RoboDK station: Estación_kuka_ibero_router.rdk

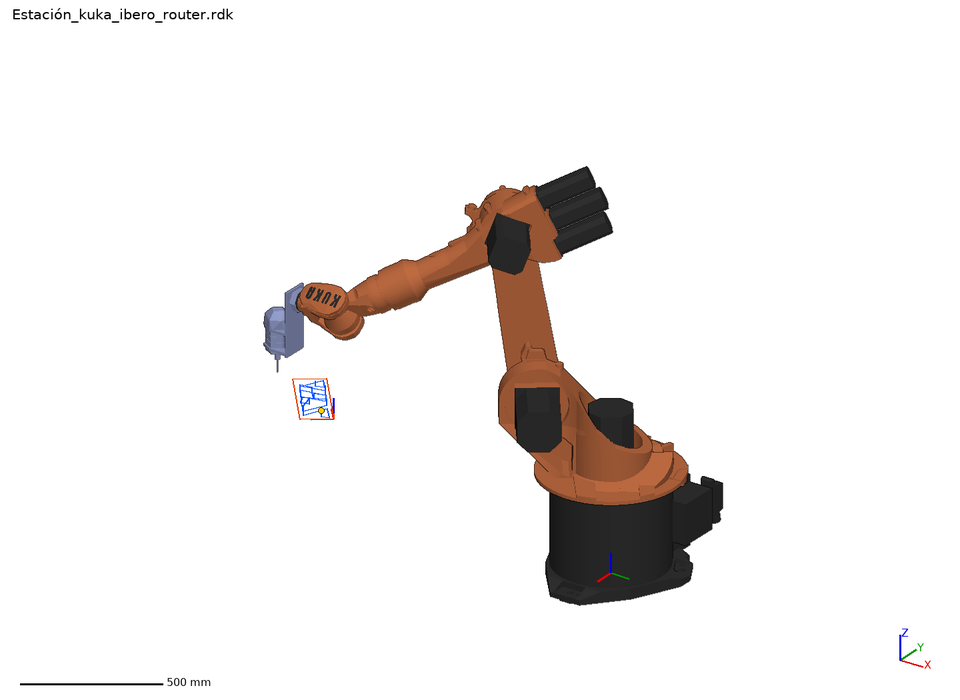
[picture v0: the station drawn from its stored meshes, robots at their saved joint values, targets as dots, program paths as lines]
Station Estación_kuka_ibero_router (saved by RoboDK 5.9.0). Poses are relative to the parent item; angles as X-Y-Z fixed-axis rotations.
Station parameters (name, value as stored): IO_5, 1, IO_2, 1
  - frame KUKA KR 16 2 Base at (0, 0, 1020) mm, rotated rx 0 ry 0 rz -90 deg
    - robot KUKA KR 16 2: 6 axes, payload 16 kg, reach 1611 mm, repeatability 0.05 mm, weight 235 kg
        modified DH rows (alpha deg, a mm, theta deg, d mm): 0, 0, 0, 675; -90, 260, 0, 0; 0, 680, -90, 0; -90, -35, 0, 670; 90, 0, 0, 0; -90, 0, 180, 158
        joint limits [-185, -155, -130, -350, -130, -350] to [185, 35, 154, 350, 130, 350]; home [0, -90, 90, 0, 0, 0]; saved at [53.134, -81.31, 105.955, 119.181, 43.406, -37.953]
      - tool Plumon_ensamble, TCP at (4.25, 1.36, 301.29) mm, size 85.6 x 85.6 x 301.8 mm, geometry from Plumon_ensamble.IGS
      - tool Ensamble_taladro, TCP at (-10.55, 304.47, 89.65) mm, rotated rx -90 ry 0 rz 0 deg, size 100 x 343.5 x 149.7 mm, geometry from Ensamble_taladro.STEP
  - object Celda_completa at (0, 0, 0) mm, size 7080 x 5029 x 2401 mm, geometry from Celda_completa.IGS
  - frame Frame 2 at (-641.11, -778.22, 1753) mm, rotated rx 0.37 ry 0.31 rz 129.33 deg
    - object Logo_jpha_3.0-Corte at (150, 150, 0) mm
  - frame Frame 3 at (-641.11, -778.23, 1751.5) mm, rotated rx 0.37 ry 0.31 rz 129.33 deg
    - object Corte_JPHA-0 at (150, 150, 0) mm
  - program O_ON (1 instructions, listed below)
  - machining project Grabado_JP: rotZ(0) | rotX(0)*rotY(0) | rotz(0) | onStart | onPathStart | onApproach | onPoint | onRetract | onFinish | SetRPM(%1) | SetTool(%1) | Extruder(%1) | default | default | OutOnMov(%1) | OutOffMov(%1) | onPathFinish | M_RunCode(%1)
  - program Grabado_JP (87 instructions, listed below)
  - machining project Corte_JP: rotZ(0) | rotX(0)*rotY(0) | rotz(0) | onStart | onPathStart | onApproach | onPoint | onRetract | onFinish | SetRPM(%1) | SetTool(%1) | Extruder(%1) | default | default | OutOnMov(%1) | OutOffMov(%1) | onPathFinish | M_RunCode(%1)
  - program Corte_JP (17 instructions, listed below)
  - program O_OFF (1 instructions, listed below)
  - program MainProgram (4 instructions, listed below)
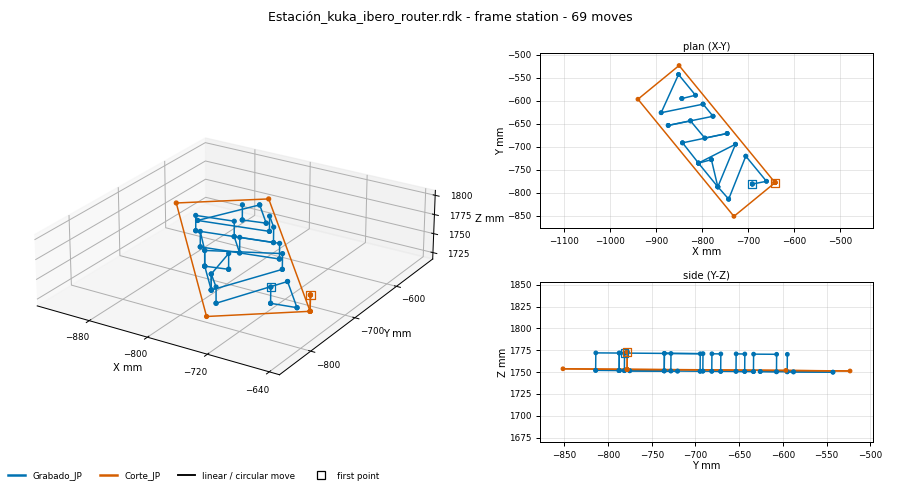
[picture p0: tool path of Estación_kuka_ibero_router.rdk in frame station, 69 of 69 moves have a stored position in this frame; points joined in program order, loops and branches not executed]

--- program O_ON (robot KUKA KR 16 2) ---
  Set IO_2=1

--- program Grabado_JP (robot KUKA KR 16 2) ---
  Suave(1)
  Establecer velocidad (1000.0 mm/s)
  Est. Ref.: Frame 3
  Est. herr: Ensamble_taladro
  Mostrar Ensamble_taladro
  MoveJ 1 to (28.97, 40.25, 20) mm, rotated rx -180 ry 0 rz -39.33 deg; joints [41.177, -79.343, 101.588, 108.422, 52.498, -29.052]
  MoveL 2 to (28.97, 40.25, 20) mm, rotated rx -180 ry 0 rz -39.33 deg; joints [41.177, -79.343, 101.588, 108.422, 52.498, -29.052]
  MoveL 3 to (28.97, 40.25, 0) mm, rotated rx 180 ry 0 rz -39.33 deg; joints [41.172, -78.564, 102.542, 109.663, 53.067, -31.108]
  MoveL 4 to (28.97, 40.25, 0) mm, rotated rx 180 ry 0 rz -39.33 deg; joints [41.172, -78.564, 102.542, 109.663, 53.067, -31.108]
  Establecer velocidad (50.0 mm/s)
  MoveL 5 to (14.16, 12.53, 0) mm, rotated rx 180 ry 0 rz -39.33 deg; joints [40.037, -80.494, 104.881, 109.228, 54.18, -31.159]
  MoveL 6 to (14.16, 12.53, 0) mm, rotated rx 180 ry 0 rz -39.33 deg; joints [40.037, -80.494, 104.881, 109.228, 54.18, -31.159]
  MoveL 7 to (85.03, 12.68, 0) mm, rotated rx 180 ry 0 rz -39.33 deg; joints [44.209, -81.297, 105.866, 112.12, 50.691, -33.064]
  MoveL 8 to (85.03, 12.68, 0) mm, rotated rx 180 ry 0 rz -39.33 deg; joints [44.209, -81.297, 105.866, 112.12, 50.691, -33.064]
  MoveL 9 to (36.22, 100.95, 0) mm, rotated rx 180 ry 0 rz -39.33 deg; joints [42.107, -74.026, 96.754, 109.349, 51.841, -29.984]
  Establecer velocidad (1000.0 mm/s)
  MoveL 10 to (36.22, 100.95, 0) mm, rotated rx 180 ry 0 rz -39.33 deg; joints [42.107, -74.026, 96.754, 109.349, 51.841, -29.984]
  MoveL 11 to (36.22, 100.95, 20) mm, rotated rx 180 ry 0 rz -39.33 deg; joints [42.112, -74.755, 95.82, 108.102, 51.303, -27.975]
  Establecer velocidad (1000.0 mm/s)
  MoveL 12 to (71.93, 102.21, 20) mm, rotated rx 180 ry 0 rz -39.33 deg; joints [44.054, -75.019, 96.177, 109.354, 49.618, -28.844]
  MoveL 13 to (71.93, 102.21, 0) mm, rotated rx -180 ry 0 rz -39.33 deg; joints [44.049, -74.286, 97.112, 110.67, 50.193, -30.89]
  MoveL 14 to (71.93, 102.21, 0) mm, rotated rx -180 ry 0 rz -39.33 deg; joints [44.049, -74.286, 97.112, 110.67, 50.193, -30.89]
  Establecer velocidad (50.0 mm/s)
  MoveL 15 to (119.27, 13.71, 0) mm, rotated rx 180 ry 0 rz -39.33 deg; joints [46.257, -81.465, 106.079, 113.618, 48.994, -34.066]
  Establecer velocidad (1000.0 mm/s)
  MoveL 16 to (119.27, 13.71, 0) mm, rotated rx 180 ry 0 rz -39.33 deg; joints [46.257, -81.465, 106.079, 113.618, 48.994, -34.066]
  MoveL 17 to (119.27, 13.71, 20) mm, rotated rx 180 ry 0 rz -39.33 deg; joints [46.263, -82.275, 105.107, 112.177, 48.295, -31.882]
  Establecer velocidad (1000.0 mm/s)
  MoveL 18 to (138.59, 102.07, 20) mm, rotated rx 180 ry 0 rz -39.33 deg; joints [47.695, -75.451, 96.766, 111.879, 46.495, -30.647]
  MoveL 19 to (138.59, 102.07, 0) mm, rotated rx -180 ry 0 rz -39.33 deg; joints [47.69, -74.714, 97.702, 113.326, 47.144, -32.763]
  MoveL 20 to (138.59, 102.07, 0) mm, rotated rx -180 ry 0 rz -39.33 deg; joints [47.69, -74.714, 97.702, 113.326, 47.144, -32.763]
  Establecer velocidad (50.0 mm/s)
  MoveL 21 to (71.93, 102.21, 0) mm, rotated rx -180 ry 0 rz -39.33 deg; joints [44.049, -74.286, 97.112, 110.67, 50.193, -30.89]
  Establecer velocidad (1000.0 mm/s)
  MoveL 22 to (71.93, 102.21, 0) mm, rotated rx -180 ry 0 rz -39.33 deg; joints [44.049, -74.286, 97.112, 110.67, 50.193, -30.89]
  MoveL 23 to (71.93, 102.21, 20) mm, rotated rx 180 ry 0 rz -39.33 deg; joints [44.054, -75.019, 96.177, 109.354, 49.618, -28.844]
  Establecer velocidad (1000.0 mm/s)
  MoveL 24 to (126.64, 75.56, 20) mm, rotated rx -180 ry 0 rz -39.33 deg; joints [46.945, -77.46, 99.309, 111.824, 47.342, -30.97]
  MoveL 25 to (126.64, 75.56, 0) mm, rotated rx 180 ry 0 rz -39.33 deg; joints [46.939, -76.7, 100.253, 113.254, 48, -33.097]
  MoveL 26 to (126.64, 75.56, 0) mm, rotated rx 180 ry 0 rz -39.33 deg; joints [46.939, -76.7, 100.253, 113.254, 48, -33.097]
  Establecer velocidad (50.0 mm/s)
  MoveL 27 to (138.59, 102.07, 0) mm, rotated rx -180 ry 0 rz -39.33 deg; joints [47.69, -74.714, 97.702, 113.326, 47.144, -32.763]
  Establecer velocidad (1000.0 mm/s)
  MoveL 28 to (138.59, 102.07, 0) mm, rotated rx -180 ry 0 rz -39.33 deg; joints [47.69, -74.714, 97.702, 113.326, 47.144, -32.763]
  MoveL 29 to (138.59, 102.07, 20) mm, rotated rx 180 ry 0 rz -39.33 deg; joints [47.695, -75.451, 96.766, 111.879, 46.495, -30.647]
  Establecer velocidad (1000.0 mm/s)
  MoveL 30 to (194.8, 100.95, 20) mm, rotated rx 180 ry 0 rz -39.33 deg; joints [50.787, -75.637, 97.032, 114.199, 43.877, -32.339]
  MoveL 31 to (194.8, 100.95, 0) mm, rotated rx 180 ry 0 rz -39.33 deg; joints [50.781, -74.897, 97.969, 115.756, 44.59, -34.515]
  MoveL 32 to (194.8, 100.95, 0) mm, rotated rx 180 ry 0 rz -39.33 deg; joints [50.781, -74.897, 97.969, 115.756, 44.59, -34.515]
  Establecer velocidad (50.0 mm/s)
  MoveL 33 to (148.94, 12.77, 0) mm, rotated rx -180 ry 0 rz -39.33 deg; joints [48.032, -81.676, 106.342, 114.992, 47.544, -35.019]
  Establecer velocidad (1000.0 mm/s)
  MoveL 34 to (148.94, 12.77, 0) mm, rotated rx -180 ry 0 rz -39.33 deg; joints [48.032, -81.676, 106.342, 114.992, 47.544, -35.019]
  MoveL 35 to (148.94, 12.77, 20) mm, rotated rx -180 ry 0 rz -39.33 deg; joints [48.038, -82.489, 105.369, 113.488, 46.806, -32.801]
  Establecer velocidad (1000.0 mm/s)
  MoveL 36 to (171.85, 56.82, 20) mm, rotated rx 180 ry 0 rz -39.33 deg; joints [49.471, -79.067, 101.316, 113.994, 45.34, -32.739]
  MoveL 37 to (171.85, 56.82, 0) mm, rotated rx 180 ry 0 rz -39.33 deg; joints [49.465, -78.29, 102.269, 115.523, 46.07, -34.931]
  MoveL 38 to (171.85, 56.82, 0) mm, rotated rx 180 ry 0 rz -39.33 deg; joints [49.465, -78.29, 102.269, 115.523, 46.07, -34.931]
  Establecer velocidad (50.0 mm/s)
  MoveL 39 to (220.8, 57.14, 0) mm, rotated rx -180 ry 0 rz -39.33 deg; joints [52.281, -78.241, 102.234, 117.838, 43.777, -36.584]
  Establecer velocidad (1000.0 mm/s)
  MoveL 40 to (220.8, 57.14, 0) mm, rotated rx -180 ry 0 rz -39.33 deg; joints [52.281, -78.241, 102.234, 117.838, 43.777, -36.584]
  MoveL 41 to (220.8, 57.14, 20) mm, rotated rx -180 ry 0 rz -39.33 deg; joints [52.287, -79.018, 101.281, 116.213, 42.986, -34.345]
  Establecer velocidad (1000.0 mm/s)
  MoveL 42 to (243.85, 100.95, 20) mm, rotated rx 180 ry 0 rz -39.33 deg; joints [53.487, -75.53, 96.92, 116.341, 41.601, -33.914]
  MoveL 43 to (243.85, 100.95, 0) mm, rotated rx 180 ry 0 rz -39.33 deg; joints [53.481, -74.79, 97.856, 117.993, 42.371, -36.139]
  MoveL 44 to (243.85, 100.95, 0) mm, rotated rx 180 ry 0 rz -39.33 deg; joints [53.481, -74.79, 97.856, 117.993, 42.371, -36.139]
  Establecer velocidad (50.0 mm/s)
  MoveL 45 to (197.51, 12.87, 0) mm, rotated rx -180 ry 0 rz -39.33 deg; joints [50.954, -81.736, 106.437, 117.36, 45.177, -36.681]
  Establecer velocidad (1000.0 mm/s)
  MoveL 46 to (197.51, 12.87, 0) mm, rotated rx -180 ry 0 rz -39.33 deg; joints [50.954, -81.736, 106.437, 117.36, 45.177, -36.681]
  MoveL 47 to (197.51, 12.87, 20) mm, rotated rx -180 ry 0 rz -39.33 deg; joints [50.961, -82.55, 105.463, 115.754, 44.372, -34.414]
  Establecer velocidad (1000.0 mm/s)
  MoveL 48 to (231.62, 12.92, 20) mm, rotated rx 180 ry 0 rz -39.33 deg; joints [53.013, -82.476, 105.396, 117.45, 42.685, -35.652]
  MoveL 49 to (231.62, 12.92, 0) mm, rotated rx -180 ry 0 rz -39.33 deg; joints [53.006, -81.663, 106.369, 119.125, 43.537, -37.949]
  MoveL 50 to (231.62, 12.92, 0) mm, rotated rx -180 ry 0 rz -39.33 deg; joints [53.006, -81.663, 106.369, 119.125, 43.537, -37.949]
  Establecer velocidad (50.0 mm/s)
  MoveL 51 to (275.08, 95.29, 0) mm, rotated rx -180 ry 0 rz -39.33 deg; joints [55.219, -75.064, 98.229, 119.638, 41.019, -37.429]
  MoveL 52 to (275.08, 95.29, 0) mm, rotated rx -180 ry 0 rz -39.33 deg; joints [55.219, -75.064, 98.229, 119.638, 41.019, -37.429]
  MoveL 53 to (315.48, 13.3, 0) mm, rotated rx 180 ry 0 rz -39.33 deg; joints [58.012, -81.056, 105.701, 123.835, 39.625, -41.449]
  MoveL 54 to (315.48, 13.3, 0) mm, rotated rx 180 ry 0 rz -39.33 deg; joints [58.012, -81.056, 105.701, 123.835, 39.625, -41.449]
  MoveL 55 to (257.09, 13.3, 0) mm, rotated rx 180 ry 0 rz -39.33 deg; joints [54.533, -81.519, 106.214, 120.494, 42.328, -38.947]
  MoveL 56 to (257.09, 13.3, 0) mm, rotated rx 180 ry 0 rz -39.33 deg; joints [54.533, -81.519, 106.214, 120.494, 42.328, -38.947]
  MoveL 57 to (270.38, 40.89, 0) mm, rotated rx 180 ry 0 rz -39.33 deg; joints [55.197, -79.285, 103.545, 120.695, 41.586, -38.847]
  Establecer velocidad (1000.0 mm/s)
  MoveL 58 to (270.38, 40.89, 0) mm, rotated rx 180 ry 0 rz -39.33 deg; joints [55.197, -79.285, 103.545, 120.695, 41.586, -38.847]
  MoveL 59 to (270.38, 40.89, 20) mm, rotated rx -180 ry 0 rz -39.33 deg; joints [55.204, -80.074, 102.587, 118.967, 40.711, -36.549]

--- program Corte_JP (robot KUKA KR 16 2) ---
  Suave(1)
  Establecer velocidad (1000.0 mm/s)
  Est. Ref.: Frame 2
  Est. herr: Ensamble_taladro
  Mostrar Ensamble_taladro
  MoveJ 1 to (0, 0, 20) mm, rotated rx 180 ry 0 rz -39.33 deg; joints [39.071, -81.996, 104.875, 107.615, 54.543, -29.055]
  MoveL 2 to (0, 0, 20) mm, rotated rx 180 ry 0 rz -39.33 deg; joints [39.071, -81.996, 104.875, 107.615, 54.543, -29.055]
  MoveL 3 to (0, 0, 0) mm, rotated rx 180 ry 0 rz -39.33 deg; joints [39.066, -81.185, 105.842, 108.803, 55.103, -31.119]
  MoveL 4 to (0, 0, 0) mm, rotated rx 180 ry 0 rz -39.33 deg; joints [39.066, -81.185, 105.842, 108.803, 55.103, -31.119]
  Establecer velocidad (50.0 mm/s)
  MoveL 5 to (0, 115.81, 0) mm, rotated rx 180 ry 0 rz -39.33 deg; joints [40.311, -72.395, 94.708, 107.954, 53.281, -28.821]
  MoveL 6 to (329.83, 115.81, 0) mm, rotated rx 180 ry 0 rz -39.33 deg; joints [58.073, -72.991, 95.672, 121.864, 38.512, -38.878]
  MoveL 7 to (329.83, 0, 0) mm, rotated rx 180 ry 0 rz -39.33 deg; joints [58.973, -81.872, 106.817, 125.143, 39.075, -42.618]
  MoveL 8 to (0, 0, 0) mm, rotated rx 180 ry 0 rz -39.33 deg; joints [39.066, -81.185, 105.842, 108.803, 55.103, -31.119]
  Establecer velocidad (1000.0 mm/s)
  MoveL 9 to (0, 0, 0) mm, rotated rx 180 ry 0 rz -39.33 deg; joints [39.066, -81.185, 105.842, 108.803, 55.103, -31.119]
  MoveL 10 to (0, 0, 20) mm, rotated rx 180 ry 0 rz -39.33 deg; joints [39.071, -81.996, 104.875, 107.615, 54.543, -29.055]

--- program O_OFF (robot KUKA KR 16 2) ---
  Set IO_2=0

--- program MainProgram (robot KUKA KR 16 2) ---
  Llamar O_ON
  Llamar Grabado_JP
  Llamar Corte_JP
  Llamar O_OFF
